FUNCTION_BLOCK JSON_FORMAT_12EFF7739F51B62A (* Generic Interface Function Block Type *)
  (* Standard: 61499-2 *)
  (* Version 0.0, 30/03/2021, SESA471728, Schneider Electric, Template *)
  PACKAGE UAO.Hackathon;
  (* Compiler Cpp nxtControl builtin 1.0 *)
  {SET_ATTRIBUTE(Runtime.FBType.ImplementingType, Runtime.Standard#DYNGEN_JSON_FORMAT)}
  {SET_ATTRIBUTE(Configuration.GenericFBType.InterfaceParams, Runtime.Base#CNT:=4;value${CNT$}:STRING,STRING,STRING,STRING)}
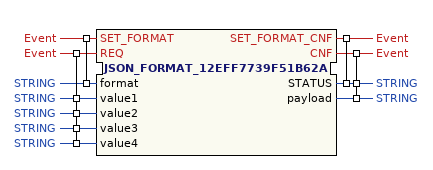
  EVENT_INPUT
    SET_FORMAT WITH format; (* Execute verification of the format *)
    REQ WITH value1, value2, value3, value4; (* Execution process *)
  END_EVENT
  EVENT_OUTPUT
    SET_FORMAT_CNF WITH STATUS; (* SET_FORMAT confirmation *)
    CNF WITH STATUS, payload; (* Execution confirmation *)
  END_EVENT
  VAR_INPUT
    format : STRING; (* JSON format *)
    value1 : STRING; (* Value *)
    value2 : STRING; (* Value *)
    value3 : STRING; (* Value *)
    value4 : STRING; (* Value *)
  END_VAR
  VAR_OUTPUT
    STATUS : STRING; (* Status *)
    payload : STRING; (* JSON payload *)
  END_VAR
  EC_STATES
    START;
  END_STATES
END_FUNCTION_BLOCK
